{attribute addProperty BoxType "EL3044-0000-0016"}
{attribute addProperty Id "AI_Standard_ChannelAT %I*ARRAY[0..24] OF AI_Standard_Channel_BC62E3BB288360WcStateAT %I*WcState_98A4DF7520.250InfoDataAT %I*InfoData_BC63D37F80100"}
{attribute addProperty CRC "1576038416"}
{attribute addProperty SizeInBites "370"}
{attribute addProperty SizeInBytes "46.25"}
TYPE EL3044_885139EF :
STRUCT
	{attribute addProperty Name "AI_Standard_Channel"}
	AI_Standard_Channel : ARRAY[0..24] OF AI_Standard_Channel_BC62E3BB;
	{attribute addProperty Name "WcState"}
	WcState : WcState_98A4DF75;
	{attribute addProperty Name "InfoData"}
	InfoData : InfoData_BC63D37F;
END_STRUCT
END_TYPE

(* stored: Version 1.2.0.0, ProductVersion 3.1.4024.9
   DUT EL3044_885139EF: Id {3e7520d5-dd9d-45c2-b3f3-6b58a525bd60} *)
